(* CoDeSys 2.3 export: IEC60870.EXP *)
(* Libraries: WagoLib60870_06.lib 28.2.20 17:12:24 *)

(* Task configuration *)
TASK IEC60870Task1 (PRIORITY := 7, INTERVAL := T#20ms);
IEC60870_MAIN_PRG
IEC60870_ServerPRG_1_104
END_TASK

(* POU IEC60870_MAIN_PRG, ST *)
PROGRAM IEC60870_MAIN_PRG
VAR_INPUT
	tonReboot			: TON := (PT := t#3s);
END_VAR
VAR
	tonSystemStart		: TON := (PT := t#1s);
END_VAR
IEC870_SyncClockOnRTC(eSyncMode := IEC870_CSM_SNTP);

(*=======================================================================================================================*)
(* Special treatment, if an reset via IEC 60870 is requested *)
tonReboot(IN := (gbyIEC870_ValueQRP = 1));
IF (tonReboot.ET < t#1s) THEN (* Normal operation *)
	;
ELSE
	IEC60870_ServerPRG_1_104.ExitAction();
	IF (tonReboot.Q) THEN
		FirmwareReset(TRUE);
	END_IF
END_IF

(*=======================================================================================================================*)
IF (gxIEC870_Enable) THEN
	IF (tonSystemStart.Q = FALSE) THEN
		(* One second after restart of the IEC 60870 application the retain variable for the cause of the restart will be reset *)
		tonSystemStart(IN := TRUE);
		gbyIEC870_RetainQRP := SEL(tonSystemStart.Q, gbyIEC870_RetainQRP, 0);
	END_IF
END_IF
END_PROGRAM

(* POU IEC870_ComHandshake, ST *)
(* Generated on: 13.10.2017 12:08:38 *)
(* IEC60870 Configurator version: 2.4.9 - 2017-04-04 *)
FUNCTION_BLOCK IEC870_ComHandshake
VAR_INPUT
	iComPort		: INT;
	pKBUS_DW		: POINTER TO ARRAY[0..1] OF WORD;
	wKBUS_ADR		: WORD;
END_VAR
VAR_OUTPUT
	xRTS			: BOOL;
	xOpen			: BOOL;
END_VAR
;
END_FUNCTION_BLOCK
ACTION ActionReadDW:
;
END_ACTION
ACTION ActionWriteDW:
;
END_ACTION
ACTION Close:
;
END_ACTION
ACTION CTS_SetHigh:
;
END_ACTION
ACTION CTS_SetLow:
;
END_ACTION
ACTION Open:
;
END_ACTION
ACTION ReadRTS:
;
END_ACTION

(* POU IEC870_ConfigTool, ST *)
(* Generated on: 13.10.2017 12:08:38 *)
(* IEC60870 Configurator version: 2.4.9 - 2017-04-04 *)
FUNCTION_BLOCK IEC870_ConfigTool
VAR_INPUT
	bEnable                     : BOOL;
	stCallString	            : STRING(250);
END_VAR
VAR_OUTPUT
	bDone			            : BOOL;
	bBusy			            : BOOL;
	stResultString	            : STRING;
	iFbResult		            : INT;
	iConfigToolResult           : INT;
	stConfigToolErrorString	    : STRING(150);
END_VAR
VAR
	fbCT				    : configToolFB;
END_VAR
fbCT(bEnable                := bEnable,
     stCallString            := stCallString,
     bDone                   => bDone,
     bBusy                   => bBusy,
     stResultString          => stResultString,
     iFbResult               => iFbResult,
     iConfigToolResult       => iConfigToolResult,
     stConfigToolErrorString => stConfigToolErrorString);
END_FUNCTION_BLOCK
